FUNCTION_BLOCK FB_ExecutionContinuity_Test EXTENDS TcUnit.FB_TestSuite
VAR done : BOOL; END_VAR

IF NOT done THEN
InitialObservationEstablishesBaseline();
ContinuousAndRepeatedCycle();
SkippedScanRequiresRecovery();
OnlineChangeDetectedWithoutGap();
TaskChangeAndInvalidContext();
CounterWrapAndReset();
CompatibleChangePreservesExecution();
CompatibleChangeCannotMaskGap();
CompatiblePolicyCannotMaskOwnerFailure();
done := TRUE; END_IF;

METHOD InitialObservationEstablishesBaseline
VAR fb : TcForge.FB_ExecutionContinuity; END_VAR
TEST('InitialObservationEstablishesBaseline');
fb(taskIndex := 1, cycleCounter := 99, onlineChangeCounter := 3); AssertFalse(Condition := fb.interrupted, Message := 'First sample establishes baseline');
TEST_FINISHED();
END_METHOD

METHOD ContinuousAndRepeatedCycle
VAR fb : TcForge.FB_ExecutionContinuity; END_VAR
TEST('ContinuousAndRepeatedCycle');
fb(taskIndex := 1, cycleCounter := 99); fb(cycleCounter := 100); AssertFalse(Condition := fb.interrupted, Message := 'Next scan continues'); fb(); AssertFalse(Condition := fb.interrupted, Message := 'Same scan observation is idempotent');
TEST_FINISHED();
END_METHOD

METHOD SkippedScanRequiresRecovery
VAR fb : TcForge.FB_ExecutionContinuity; END_VAR
TEST('SkippedScanRequiresRecovery');
fb(taskIndex := 1, cycleCounter := 99); fb(cycleCounter := 101); AssertTrue(Condition := fb.interrupted, Message := 'Missed execution detected'); fb(cycleCounter := 102); AssertFalse(Condition := fb.interrupted, Message := 'Caller must latch recovery; event is one scan');
TEST_FINISHED();
END_METHOD

METHOD OnlineChangeDetectedWithoutGap
VAR fb : TcForge.FB_ExecutionContinuity; END_VAR
TEST('OnlineChangeDetectedWithoutGap');
fb(taskIndex := 1, cycleCounter := 99, onlineChangeCounter := 3); fb(cycleCounter := 100, onlineChangeCounter := 4); AssertTrue(Condition := fb.interrupted, Message := 'Implementation-only online change detected');
TEST_FINISHED();
END_METHOD

METHOD TaskChangeAndInvalidContext
VAR fb : TcForge.FB_ExecutionContinuity; END_VAR
TEST('TaskChangeAndInvalidContext');
fb(taskIndex := 1, cycleCounter := 99); fb(taskIndex := 2, cycleCounter := 100); AssertTrue(Condition := fb.interrupted, Message := 'Different owner detected'); fb(taskIndex := 0); AssertTrue(Condition := fb.interrupted, Message := 'RPC or invalid context rejected');
TEST_FINISHED();
END_METHOD

METHOD CounterWrapAndReset
VAR fb : TcForge.FB_ExecutionContinuity; END_VAR
TEST('CounterWrapAndReset');
fb(taskIndex := 1, cycleCounter := UDINT#16#FFFFFFFF); fb(cycleCounter := 0); AssertFalse(Condition := fb.interrupted, Message := 'Natural wrap is continuous'); fb(cycleCounter := 99); fb(cycleCounter := 0); AssertTrue(Condition := fb.interrupted, Message := 'Counter discontinuity detected');
TEST_FINISHED();
END_METHOD

METHOD CompatibleChangePreservesExecution
VAR fb : TcForge.FB_ExecutionContinuity; END_VAR
TEST('CompatibleChangePreservesExecution');
fb(taskIndex := 1, cycleCounter := 99, onlineChangeCounter := 3, recoverOnOnlineChange := FALSE);
fb(cycleCounter := 100, onlineChangeCounter := 4);
AssertTrue(Condition := fb.onlineChanged, Message := 'Change remains observable');
AssertFalse(Condition := fb.executionInterrupted, Message := 'Online edit is not an execution gap');
AssertFalse(Condition := fb.interrupted, Message := 'Explicit compatible-edit policy preserves execution');
fb(cycleCounter := 101);
AssertFalse(Condition := fb.onlineChanged, Message := 'Change notification is a pulse');
TEST_FINISHED();
END_METHOD

METHOD CompatibleChangeCannotMaskGap
VAR fb : TcForge.FB_ExecutionContinuity; END_VAR
TEST('CompatibleChangeCannotMaskGap');
fb(taskIndex := 1, cycleCounter := 99, onlineChangeCounter := 3, recoverOnOnlineChange := FALSE);
fb(cycleCounter := 101, onlineChangeCounter := 4);
AssertTrue(Condition := fb.onlineChanged, Message := 'Simultaneous online edit observed');
AssertTrue(Condition := fb.executionInterrupted, Message := 'Gap remains a gap during online edit');
AssertTrue(Condition := fb.interrupted, Message := 'Compatible-edit policy cannot suppress recovery');
TEST_FINISHED();
END_METHOD

METHOD CompatiblePolicyCannotMaskOwnerFailure
VAR fb : TcForge.FB_ExecutionContinuity; END_VAR
TEST('CompatiblePolicyCannotMaskOwnerFailure');
fb(taskIndex := 1, cycleCounter := 99, recoverOnOnlineChange := FALSE);
fb(taskIndex := 2, cycleCounter := 100);
AssertTrue(Condition := fb.interrupted, Message := 'Owner conflict still requires recovery');
fb(taskIndex := 0);
AssertTrue(Condition := fb.executionInterrupted, Message := 'Invalid context still fails closed');
TEST_FINISHED();
END_METHOD

END_FUNCTION_BLOCK

(* stored: Version 1.1.0.1
   POU FB_ExecutionContinuity_Test: Id {f666fe2e-1149-484e-bbf4-abaa632eaebf}
   Method InitialObservationEstablishesBaseline: Id {fd637c91-5d4c-474f-9b62-53c01240f01f}
   Method ContinuousAndRepeatedCycle: Id {8e0acbee-e5b2-4100-aa22-230cddb46ef5}
   Method SkippedScanRequiresRecovery: Id {ca528c56-5566-4a21-9a75-89c0945e6e1b}
   Method OnlineChangeDetectedWithoutGap: Id {5dcf1065-db81-42e2-897d-02f125642727}
   Method TaskChangeAndInvalidContext: Id {bf3b21da-8dd2-4b8b-9378-f36750e8674d}
   Method CounterWrapAndReset: Id {5a54f69c-7298-4ef0-9f2e-22778f2caecd}
   Method CompatibleChangePreservesExecution: Id {985ce2be-8e0d-4375-b688-a5d00b13cba2}
   Method CompatibleChangeCannotMaskGap: Id {7ee05729-d075-40ba-9c1f-b3af6d45b09e}
   Method CompatiblePolicyCannotMaskOwnerFailure: Id {e7723f75-2354-47e4-a5e1-12d2b1911e61} *)
